FUNCTION SPLITTING_DWORD_INTO_QUARTERS
  (* Standard: 61499-1; Description: Copyright (c) 2024 HR Agrartechnik GmbH This program and the accompanying materials are made available under the terms of the Eclipse Public License 2.0 which is available at https://www.eclipse.org/legal/epl-2.0/ SPDX-License-Identifier: EPL-2.0 *)
  (* Version 1.0, 2024-02-22, franz *)
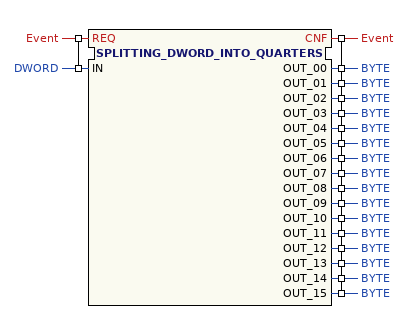
  EVENT_INPUT
    REQ WITH IN; (* Normal Execution Request *)
  END_EVENT
  EVENT_OUTPUT
    CNF WITH OUT_00, OUT_01, OUT_02, OUT_03, OUT_04, OUT_05, OUT_06, OUT_07, OUT_08, OUT_09, OUT_10, OUT_11, OUT_12, OUT_13, OUT_14, OUT_15; (* Execution Confirmation *)
  END_EVENT
  VAR_INPUT
    IN : DWORD; (* DWORD Input *)
  END_VAR
  VAR_OUTPUT
    OUT_00 : BYTE; (* QUARTER BYTE 00 *)
    OUT_01 : BYTE; (* QUARTER BYTE 01 *)
    OUT_02 : BYTE; (* QUARTER BYTE 02 *)
    OUT_03 : BYTE; (* QUARTER BYTE 03 *)
    OUT_04 : BYTE; (* QUARTER BYTE 04 *)
    OUT_05 : BYTE; (* QUARTER BYTE 05 *)
    OUT_06 : BYTE; (* QUARTER BYTE 06 *)
    OUT_07 : BYTE; (* QUARTER BYTE 07 *)
    OUT_08 : BYTE; (* QUARTER BYTE 08 *)
    OUT_09 : BYTE; (* QUARTER BYTE 09 *)
    OUT_10 : BYTE; (* QUARTER BYTE 10 *)
    OUT_11 : BYTE; (* QUARTER BYTE 11 *)
    OUT_12 : BYTE; (* QUARTER BYTE 12 *)
    OUT_13 : BYTE; (* QUARTER BYTE 13 *)
    OUT_14 : BYTE; (* QUARTER BYTE 14 *)
    OUT_15 : BYTE; (* QUARTER BYTE 15 *)
  END_VAR
  BODY IN ST:
FUNCTION SPLITTING_DWORD_INTO_QUARTERS

VAR_INPUT
	IN : DWORD;    // DWORD Input
END_VAR

VAR_OUTPUT
	OUT_00 : BYTE;    // QUARTER BYTE 00
	OUT_01 : BYTE;    // QUARTER BYTE 01
	OUT_02 : BYTE;    // QUARTER BYTE 02
	OUT_03 : BYTE;    // QUARTER BYTE 03
	OUT_04 : BYTE;    // QUARTER BYTE 04
	OUT_05 : BYTE;    // QUARTER BYTE 05
	OUT_06 : BYTE;    // QUARTER BYTE 06
	OUT_07 : BYTE;    // QUARTER BYTE 07
	OUT_08 : BYTE;    // QUARTER BYTE 08
	OUT_09 : BYTE;    // QUARTER BYTE 09
	OUT_10 : BYTE;    // QUARTER BYTE 10
	OUT_11 : BYTE;    // QUARTER BYTE 11
	OUT_12 : BYTE;    // QUARTER BYTE 12
	OUT_13 : BYTE;    // QUARTER BYTE 13
	OUT_14 : BYTE;    // QUARTER BYTE 14
	OUT_15 : BYTE;    // QUARTER BYTE 15
END_VAR

(* this Function extracts the 16 QUARTER BYTE from a dword *)
OUT_00 := DWORD_TO_BYTE(SHR(IN AND DWORD_QUARTER_00, SHFT_QUARTER_00));
OUT_01 := DWORD_TO_BYTE(SHR(IN AND DWORD_QUARTER_01, SHFT_QUARTER_01));
OUT_02 := DWORD_TO_BYTE(SHR(IN AND DWORD_QUARTER_02, SHFT_QUARTER_02));
OUT_03 := DWORD_TO_BYTE(SHR(IN AND DWORD_QUARTER_03, SHFT_QUARTER_03));
OUT_04 := DWORD_TO_BYTE(SHR(IN AND DWORD_QUARTER_04, SHFT_QUARTER_04));
OUT_05 := DWORD_TO_BYTE(SHR(IN AND DWORD_QUARTER_05, SHFT_QUARTER_05));
OUT_06 := DWORD_TO_BYTE(SHR(IN AND DWORD_QUARTER_06, SHFT_QUARTER_06));
OUT_07 := DWORD_TO_BYTE(SHR(IN AND DWORD_QUARTER_07, SHFT_QUARTER_07));
OUT_08 := DWORD_TO_BYTE(SHR(IN AND DWORD_QUARTER_08, SHIFT_QUARTER_08));
OUT_09 := DWORD_TO_BYTE(SHR(IN AND DWORD_QUARTER_09, SHIFT_QUARTER_09));
OUT_10 := DWORD_TO_BYTE(SHR(IN AND DWORD_QUARTER_10, SHIFT_QUARTER_10));
OUT_11 := DWORD_TO_BYTE(SHR(IN AND DWORD_QUARTER_11, SHIFT_QUARTER_11));
OUT_12 := DWORD_TO_BYTE(SHR(IN AND DWORD_QUARTER_12, SHIFT_QUARTER_12));
OUT_13 := DWORD_TO_BYTE(SHR(IN AND DWORD_QUARTER_13, SHIFT_QUARTER_13));
OUT_14 := DWORD_TO_BYTE(SHR(IN AND DWORD_QUARTER_14, SHIFT_QUARTER_14));
OUT_15 := DWORD_TO_BYTE(SHR(IN AND DWORD_QUARTER_15, SHIFT_QUARTER_15));
END_FUNCTION
  END_BODY
END_FUNCTION
